FUNCTION_BLOCK FB_EQ2HOR2
VAR_INPUT
	// right ascension in degrees
	alpha: LREAL;
	// declination in degrees
	delta: LREAL;
	// longitude in degrees
	lon: LREAL;
	// latitude in degrees
	lat: LREAL;
	// Julian Days
	JD: LREAL;
END_VAR
VAR_OUTPUT
	// altitude in degrees
	alt: LREAL;
	// azimuth in degrees
	az: LREAL;
	// hour angle in degreesss
	ha: LREAL;
END_VAR
VAR
	lst, 
	T , theta0, gmst: LREAL;
	sinalt, sinaz, cosaz, az2: LREAL;
END_VAR
VAR CONSTANT
	d2r:	LREAL := PI/180.0;
	r2d:	LREAL := 180.0/PI;
	h2r:	LREAL := PI/12.0;
	h2d:	LREAL := 15.0;
END_VAR

(* 
source: http://star-www.st-and.ac.uk/~fv/webnotes/chapter7.htm
https://squarewidget.com/astronomical-calculations-sidereal-time/

*)
//lst := ct2lst(lon, jd);
T := ((JD - 2451545.0) / 36525);
theta0 := 280.46061837 + 360.98564736629 * (JD - 2451545.0) + (0.000387933 * T * T) - (T * T * T / 38710000.0); // (12.4)
gmst := MODABS(theta0, 360.0);
lst := gmst + lon; // LST in degrees
// ha := MODABS(lst*15.0 - alpha, 360.0);
ha := MODABS(lst - alpha, 360.0);
sinalt := (SIN(delta*d2r)*SIN(lat*d2r)) + (COS(delta*d2r)*COS(lat*d2r)*COS(ha*d2r));
alt := ASIN(sinalt) * r2d;

sinaz := -SIN(ha*d2r)*COS(delta*d2r)/COS(alt*d2r);
//az := ASIN(sinaz) * r2d;
az := MODABS((360 + ASIN(sinaz) * r2d), 360.0);

cosaz := (SIN(delta*d2r) - SIN(lat*d2r)*sinalt)/(COS(lat*d2r)*COS(alt*d2r));
az2 := ACOS(cosaz) * r2d;

END_FUNCTION_BLOCK

(* stored: Version 1.1.0.1, ProductVersion 3.1.4024.6
   POU FB_EQ2HOR2: Id {7b34f02a-1435-4300-8153-5c49f62d1b5b}, SpecialFunc None *)
